# EPICS substitutions: ek9000App/Db/EL4002.substitutions
file EL4002.template
{       pattern
        {
                TERMINAL,

        }
        {
        }
}
